ABB RobotStudio station: practica_2_sys_ref.rsstnx

Station practica_2_sys_ref (saved by RobotStudio 24.3.10885.0)
Controller Controlador1, task T_ROB1: task frame (RAPID world) sits at (735.42, -472.81, 500) mm in the station
Controller Controlador1
  mechanical unit ROB_1: IRB120_3_58__01, 6 joints, base frame (-735.42, 472.81, 0) mm
Layout (positions relative to the parent item):
  - IRB120_3_58__01 [mechanism, from %ABB.RobotStudio.Models.IRB120%\IRB120_3_58_G_01.rslib] at (0, 0, 500) mm; joint values [0.016, 0.6741, -0.685, -2.3981, 0.0236, 2.3978] (rad or m)
  - Pieza_1 [part] at (250, 200, 10) mm, rotated rx 0 ry 0 rz 90 deg, size 20 x 30 x 20 mm
  - Pieza_3 [part], size 500 x 400 x 10 mm
  - Sistema de coordenadas_2 [frame]
Targets, tools, work objects and paths stored in the station, written as RAPID:
! task T_ROB1
MODULE CalibData
  TASK PERS wobjdata WO_1:=[FALSE,TRUE,"",[[-735.416,472.807,-490],[1,0,0,0]],[[235,190,0],[1,0,0,0]]];
ENDMODULE

